(* PLC project Tc2_Utilities.PLC_Reset Demo, tc3-libraries-kb TwinCAT 3.1 *)
(* stored: creationDateTime 2026-05-10T20:00:00, modificationDateTime 2026-05-10T20:00:00 *)

PROGRAM P_Demo_PLC_Reset
  VAR
    fbPLC_Reset : PLC_Reset;  (* Tc2_Utilities.PLC_Reset 实例 *)
    arg_NETID : T_AmsNetId;  (* VAR_INPUT NETID *)
    arg_PORT : T_AmsPort;  (* VAR_INPUT PORT *)
    arg_RESET : BOOL;  (* VAR_INPUT RESET *)
    arg_TMOUT : TIME;  (* VAR_INPUT TMOUT *)
    out_BUSY : BOOL;  (* VAR_OUTPUT BUSY *)
    out_ERR : BOOL;  (* VAR_OUTPUT ERR *)
    out_ERRID : UDINT;  (* VAR_OUTPUT ERRID *)
  END_VAR

            // ============================================================
// Tc2_Utilities.PLC_Reset 演示程序（FB 实例）
// ============================================================
// 验证步骤：
//   1. 引用 Tc2_Utilities（及依赖类型所在库 Tc2_System 等）
//   2. 编译 + 登录
//   3. 按 doc.md 给 arg_* 赋值
//   4. 在线监视 out_* / io_* 输出
// ============================================================

fbPLC_Reset(
    NETID := arg_NETID,
    PORT := arg_PORT,
    RESET := arg_RESET,
    TMOUT := arg_TMOUT,
    BUSY => out_BUSY,
    ERR => out_ERR,
    ERRID => out_ERRID
);

          
END_PROGRAM
